TYPE ST_Test :
STRUCT
	nByte: BYTE;
	fReal: REAL;
	iSint: SINT;
	tTime: TIME;
	arrString: ARRAY[1..5] OF STRING(6);
	iInt: INT;
END_STRUCT
END_TYPE

(* stored: Version 1.1.0.1, ProductVersion 3.1.0.36
   DUT ST_Test: Id {2572a3c2-780d-4fbd-bde2-30ae7d899270} *)
